{attribute addProperty BoxType "EL2535-0000-0016"}
{attribute addProperty Id "ControlAT %Q*Control_C38C93251621PWM_outputAT %Q*INT16217"}
{attribute addProperty CRC "624683617"}
{attribute addProperty SizeInBites "32"}
{attribute addProperty SizeInBytes "4"}
TYPE PWM_Control_Channel_253BEA61 :
STRUCT
	{attribute addProperty Name "Control"}
	Control AT %Q* : Control_C38C9325;
	{attribute addProperty Name "PWM_output"}
	PWM_output AT %Q* : INT;
END_STRUCT
END_TYPE

(* stored: Version 1.2.0.0, ProductVersion 3.1.4024.9
   DUT PWM_Control_Channel_253BEA61: Id {2650ada0-88bd-4793-86bc-9ed52a2bee8f} *)
